PROGRAM PG_Besucher
VAR
	FB_Besucher_0: FB_Besucher;
END_VAR

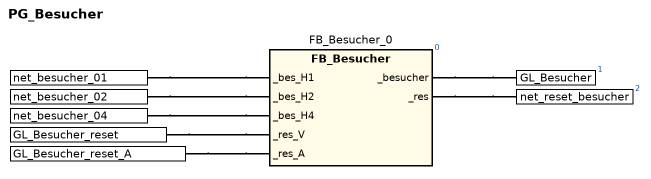
FB_Besucher_0(
    _bes_H1 := net_besucher_01,
    _bes_H2 := net_besucher_02,
    _bes_H4 := net_besucher_04,
    _res_V := GL_Besucher_reset,
    _res_A := GL_Besucher_reset_A); // FB_Besucher
GL_Besucher := FB_Besucher_0._besucher;
net_reset_besucher := FB_Besucher_0._res;

END_PROGRAM

(* stored: Version 1.1.0.1, ProductVersion 3.1.4018.5
   POU PG_Besucher: Id {e3b8a431-d0a2-4517-889e-4cfb5d991cbb}, SpecialFunc None *)
